TYPE E_OdriveInputMode :
(
    Inactive := 0,
    Passthrough := 1,
    VelRamp := 2,
    PosFilter := 3,
    //MixChannels := 4,
    TrapTraj := 5
    //TorqueRamp := 6,
    //Mirror := 7,
    //Tuning := 8
) UDINT;
END_TYPE

(* stored: Version 1.1.0.1
   DUT E_OdriveInputMode: Id {95a2bdb4-0c44-4852-9860-0786856c9726} *)
